FUNCTION_BLOCK AxesRotationAxisWidget
VAR_INPUT
    activeTab : AxesRotationAxisTabs;
    axisTitle : STRING;
    driveChannelTitle : STRING;
END_VAR
VAR_OUTPUT
END_VAR
VAR_IN_OUT
    ref : AxesRotationAxis;
    ref_driveChannel : AX52XXDriveChannel;
END_VAR
VAR
	actualStatus : StatusWidget;
    
    processes_powerOnStatus : StatusWidget;
    processes_powerOffStatus : StatusWidget;
    processes_resetStatus : StatusWidget;
    processes_stopStatus : StatusWidget;
    processes_moveAbsoluteStatus : StatusWidget;
    processes_moveRelativeStatus : StatusWidget;
    processes_moveVelocityStatus : StatusWidget;
    processes_moveOutOfLimitSwitchStatus : StatusWidget;
    
    processCommonHealthStatus : HealthStatus;
    processCommonBusyStatus   : BusyStatus;
    processCommonStatusColor  : StatusColor;
    
    
    button_overview         : SubSubSystemButtonWidget('Overview'           , AxesRotationAxisTabs.OVERVIEW);
    button_processes        : SubSubSystemButtonWidget('Processes'          , AxesRotationAxisTabs.PROCESSES);
    button_driveChannel     : SubSubSystemButtonWidget('Drive channel'      , AxesRotationAxisTabs.DRIVE_CHANNEL);   
    button_virtualAxis      : SubSubSystemButtonWidget('Virtual axis'       , AxesRotationAxisTabs.VIRTUAL_AXIS);  
    button_physicalAxis     : SubSubSystemButtonWidget('Physical axis'      , AxesRotationAxisTabs.PHYSICAL_AXIS);  
    
    driveChannel    : AX52XXDriveChannelWidget;
    virtualAxis     : AngularAxisWidget;
    physicalAxis    : AngularAxisWidget;
    
    
    actPos : AxesAngleWidget;
    setPos : AxesAngleWidget;
    targetPos : AxesAngleWidget;
END_VAR


actualStatus(text  := ref.actualStatus,
             color := HealthBusyToColor(healthStatus := ref.statuses.healthStatus, 
                                        busyStatus   := ref.statuses.busyStatus));

processes_powerOffStatus(
    text  := ref.processes.powerOff.actualStatus,
    color := HealthBusyToColor(healthStatus := ref.processes.powerOff.statuses.healthStatus, 
                               busyStatus   := ref.processes.powerOff.statuses.busyStatus));
processes_powerOnStatus(
    text  := ref.processes.powerOn.actualStatus,
    color := HealthBusyToColor(healthStatus := ref.processes.powerOn.statuses.healthStatus, 
                               busyStatus   := ref.processes.powerOn.statuses.busyStatus));
processes_resetStatus(
    text  := ref.processes.reset.actualStatus,
    color := HealthBusyToColor(healthStatus := ref.processes.reset.statuses.healthStatus, 
                               busyStatus   := ref.processes.reset.statuses.busyStatus));
processes_stopStatus(
    text  := ref.processes.stop.actualStatus,
    color := HealthBusyToColor(healthStatus := ref.processes.stop.statuses.healthStatus, 
                               busyStatus   := ref.processes.stop.statuses.busyStatus));
processes_moveAbsoluteStatus(
    text  := ref.processes.moveAbsolute.actualStatus,
    color := HealthBusyToColor(healthStatus := ref.processes.moveAbsolute.statuses.healthStatus, 
                               busyStatus   := ref.processes.moveAbsolute.statuses.busyStatus));
processes_moveRelativeStatus(
    text  := ref.processes.moveRelative.actualStatus,
    color := HealthBusyToColor(healthStatus := ref.processes.moveRelative.statuses.healthStatus, 
                               busyStatus   := ref.processes.moveRelative.statuses.busyStatus));
processes_moveVelocityStatus(
    text  := ref.processes.moveVelocity.actualStatus,
    color := HealthBusyToColor(healthStatus := ref.processes.moveVelocity.statuses.healthStatus, 
                               busyStatus   := ref.processes.moveVelocity.statuses.busyStatus));
processes_moveOutOfLimitSwitchStatus(
    text  := ref.processes.moveOutOfLimitSwitch.actualStatus,
    color := HealthBusyToColor(healthStatus := ref.processes.moveOutOfLimitSwitch.statuses.healthStatus, 
                               busyStatus   := ref.processes.moveOutOfLimitSwitch.statuses.busyStatus));

driveChannel(ref := ref_driveChannel, name := driveChannelTitle);
virtualAxis(baseRef := ref.parts.virtualAxis, ref := ref.parts.virtualAxis);
physicalAxis(baseRef := ref.parts.physicalAxis, ref := ref.parts.physicalAxis);                

processCommonHealthStatus(
     isGood :=      ref.processes.powerOn.statuses.healthStatus.isGood 
                AND ref.processes.powerOff.statuses.healthStatus.isGood
                AND ref.processes.reset.statuses.healthStatus.isGood
                AND ref.processes.stop.statuses.healthStatus.isGood
                AND ref.processes.moveAbsolute.statuses.healthStatus.isGood
                AND ref.processes.moveRelative.statuses.healthStatus.isGood
                AND ref.processes.moveVelocity.statuses.healthStatus.isGood
                AND ref.processes.moveOutOfLimitSwitch.statuses.healthStatus.isGood,
     hasWarning :=  ref.processes.powerOn.statuses.healthStatus.hasWarning 
                 OR ref.processes.powerOff.statuses.healthStatus.hasWarning
                 OR ref.processes.reset.statuses.healthStatus.hasWarning
                 OR ref.processes.stop.statuses.healthStatus.hasWarning
                 OR ref.processes.moveAbsolute.statuses.healthStatus.hasWarning
                 OR ref.processes.moveRelative.statuses.healthStatus.hasWarning
                 OR ref.processes.moveVelocity.statuses.healthStatus.hasWarning
                 OR ref.processes.moveOutOfLimitSwitch.statuses.healthStatus.hasWarning);

processCommonBusyStatus(
    isBusy :=      ref.processes.powerOn.statuses.busyStatus.busy 
                 OR ref.processes.powerOff.statuses.busyStatus.busy
                 OR ref.processes.reset.statuses.busyStatus.busy
                 OR ref.processes.stop.statuses.busyStatus.busy
                 OR ref.processes.moveAbsolute.statuses.busyStatus.busy
                 OR ref.processes.moveRelative.statuses.busyStatus.busy
                 OR ref.processes.moveVelocity.statuses.busyStatus.busy
                 OR ref.processes.moveOutOfLimitSwitch.statuses.busyStatus.busy);

processCommonStatusColor := HealthBusyToColor(healthStatus := processCommonHealthStatus, busyStatus := processCommonBusyStatus);

button_overview(        color := actualStatus.color                     , activeTab := activeTab);
button_processes(       color := processCommonStatusColor               , activeTab := activeTab);
button_driveChannel(    color := driveChannel.actualStatus.color        , activeTab := activeTab);
button_virtualAxis(     color := virtualAxis.base.actualStatus.color    , activeTab := activeTab);
button_physicalAxis(    color := physicalAxis.base.actualStatus.color   , activeTab := activeTab);

actPos(degrees := ref.actPos.degrees.value, format := '%d° %.2d$' %04.1f"', showPlus := FALSE, showMinus := TRUE);
setPos(degrees := ref.setPos.degrees.value, format := '%d° %.2d$' %04.1f"', showPlus := FALSE, showMinus := TRUE);
targetPos(degrees := ref.targetPos.degrees.value, format := '%d° %.2d$' %04.1f"', showPlus := FALSE, showMinus := TRUE);

END_FUNCTION_BLOCK

(* stored: Version 1.1.0.1, ProductVersion 3.1.4019.2
   POU AxesRotationAxisWidget: Id {732eb8b9-8b7a-472e-8af7-8ff4bc76ec04}, SpecialFunc None *)
